Fanuc KAREL source: ka00068.KL

-- PROVISIONAL review KL for V1013-1; original PC SHA256 9f681985374ac2a74064fa8cbd7f70a157341ca3dee8264f92176d81905a5be8
-- Incomplete behavior may be omitted. Consult companion uncertainty JSON. Do not deploy.
PROGRAM KA00068
%NOLOCKGROUP
-- UNRESOLVED_DECL SRC type=000102
-- UNRESOLVED_DECL DST type=000199
BEGIN
  -- UNRESOLVED_PC offsets 5-20; opcodes 2E,22,32,35
  -- UNRESOLVED_PC offsets 25-45; opcodes 49,7E,4A
  -- UNRESOLVED_PC offsets 50-54; opcodes 7F
END KA00068
